// TIA Portal V15.1 export
// export: Created 2026-01-09T13:45:14.0664329Z, ExportSetting WithDefaults, WithReadOnly, DisplayName Totally Integrated Automation Portal, DisplayVersion V15.1 Update 8, DisplayName TIA Portal Openness, DisplayVersion V15.1 Update 8, DisplayName STEP 7 Professional, DisplayVersion V15.1 Update 8, DisplayName WinCC Advanced, DisplayVersion V15.1 Update 8
DATA_BLOCK "C#2_WB"   // DB2
{ S7_Optimized_Access := 'FALSE' }
VERSION : 0.1
// stored: AutoNumber true, CodeModifiedDate 2026-01-04T14:05:19.1281212Z, CompileDate 2026-01-04T14:27:04.768919Z, CreationDate 2024-10-12T12:36:08.0193576Z, DBAccessibleFromOPCUA true, InterfaceModifiedDate 2026-01-04T14:05:19.1281212Z, IsConsistent true, IsKnowHowProtected false, IsOnlyStoredInLoadMemory false, IsPLCDB false, IsWriteProtectedInAS false, ModifiedDate 2026-01-04T14:05:19.1281212Z, ParameterModified 2026-01-04T14:05:19.1281212Z, StructureModified 2026-01-04T14:05:19.1281212Z
   VAR
      F1_NN_RUN : Bool;   // F1 Nút nhấn chạy
      F2_SW_PAU : Bool;   // F2 Công tắc tạm dừng
      F3_NN_STOP : Bool;   // F3 Nút nhấn dừng/hủy mẻ
      F4_SW_SIM : Bool;   // F4 Công tắc chế độ mô phỏng
      "SW_MAN/AUTO" : Bool;   // Công tắc chế độ chạy tay/tự động
      SW_XA_LIEU : Bool;   // Công tắc chế độ xả cân cốt liệu
      SW_NAP_NOI_TRON : Bool;   // Công tắc nạp liệu nồi trộn
      SW_XA_NOI_TRON : Bool;   // Công tắc chế độ xả bê tông
      "NN_NOI TRON" : Bool;   // Nút nhấn Nồi trộn
      NN_BTX : Bool;   // Nút nhấn Băng tải xiên
      NN_BTN : Bool;   // Nút nhấn Băng tải ngang
      "NN_TANG SAY" : Bool;   // Nút nhấn Tang sấy cốt liệu
      "NN_BOM DAU" : Bool;   // Nút nhấn Bơm dầu DO
      "NN_GAU COT LIEU" : Bool;   // Nút nhấn Gàu tải cốt liệu nóng
      "NN_SAN RUNG" : Bool;   // Nút nhấn Sàn rung cốt liệu
      "NN_GAU FD" : Bool;   // Nút nhấn Gàu tải phụ F/D
      "NN_VIT TAI FD" : Bool;   // Nút nhấn Vít tải F/D
      "NN_BOM SBS" : Bool;   // Nút nhấn Bơm nạp hạt nhựa SBS
      "NN_QUAT GIO" : Bool;   // Nút nhấn Quạt gió lọc bụi
      "NN_BOM NUOC" : Bool;   // Nút nhấn Bơm nước lọc bụi
      "NN_MO CUA" : Bool;   // Nút nhấn Van mở cửa nồi trộn
      "NN_DONG CUA" : Bool;   // Nút nhấn Van đóng cửa nồi trộn
      NN_MNK : Bool;   // Nút nhấn Máy nén khí
      "SW_XA CL1" : Bool;   // Công tắc Băng tải xả cốt liệu 1
      "SW_XA CL2" : Bool;   // Công tắc Băng tải xả cốt liệu 2
      "SW_XA CL3" : Bool;   // Công tắc Băng tải xả cốt liệu 3
      "SW_XA CL4" : Bool;   // Công tắc Băng tải xả cốt liệu 4
      "SW_XA CL5" : Bool;   // Công tắc Băng tải xả cốt liệu 5
      "NN_CAN AG1" : Bool;   // Nút nhấn Van cân AG1
      "NN_CAN AG2" : Bool;   // Nút nhấn Van cân AG2
      "NN_CAN AG3" : Bool;   // Nút nhấn Van cân AG3
      "NN_CAN AG4" : Bool;   // Nút nhấn Van cân AG4
      "NN_CAN AG5" : Bool;   // Nút nhấn Van cân AG5
      "NN_CAN FD1" : Bool;   // Nút nhấn Van cân F/D
      "NN_CAN AP1" : Bool;   // Nút nhấn Bơm nhựa
      "NN_CAN SB1" : Bool;   // Nút nhấn Van cân hạt nhựa SBS
      "SW_XA W_AG1" : Bool;   // Công tắc Van xả cân AG1
      "SW_XA W_FD1" : Bool;   // Công tắc Van xả cân FD1
      "SW_XA W_AP1" : Bool;   // Công tắc Van xả cân AP1
      "SW_XA W_SB1" : Bool;   // Công tắc Van xả cân SB1
      "NN_BOM TUOI NHUA" : Bool;   // Nút nhấn Bổ sung 1
      "NN_XA HET AGG" : Bool;   // Nút nhấn Bổ sung 2
      "NN_DAU DOT" : Bool;   // Nút nhấn Bổ sung 3
      NN_VAN_PNSBS : Bool;   // Nút nhấn Bổ sung 4
      "NN_NOTE 5" : Bool;   // Nút nhấn Bổ sung 5
      "NN_NOTE 6" : Bool;   // Nút nhấn Bổ sung 6
      "NN_NOTE 7" : Bool;   // Nút nhấn Bổ sung 7
      NN_FU_AG1 : Bool;   // Nút nhấn Báo đầy silo AG1
      NN_FU_AG2 : Bool;   // Nút nhấn Báo đầy silo AG2
      NN_FU_AG3 : Bool;   // Nút nhấn Báo đầy silo AG3
      NN_FU_AG4 : Bool;   // Nút nhấn Báo đầy silo AG4
      NN_FU_AG5 : Bool;   // Nút nhấn Báo đầy silo AG5
      NN_FU_FD1 : Bool;   // Nút nhấn Báo đầy silo FD1
      NN_FU_AP1 : Bool;   // Nút nhấn Báo đầy silo AP1
      NN_FU_SB1 : Bool;   // Nút nhấn Báo đầy silo SBS1
      SW_PA_AG1 : Bool;   // Công tắc Tạm dừng cân AG1
      SW_PA_AG2 : Bool;   // Công tắc Tạm dừng cân AG2
      SW_PA_AG3 : Bool;   // Công tắc Tạm dừng cân AG3
      SW_PA_AG4 : Bool;   // Công tắc Tạm dừng cân AG4
      SW_PA_AG5 : Bool;   // Công tắc Tạm dừng cân AG5
      SW_PA_FD1 : Bool;   // Công tắc Tạm dừng cân FD1
      SW_PA_AP1 : Bool;   // Công tắc Tạm dừng cân AP1
      SW_PA_SB1 : Bool;   // Công tắc Tạm dừng cân SBS1
      NN_ZERO_AG1 : Bool;   // Nút nhấn chỉnh 0 cân AG1
      NN_SPAN_AG1 : Bool;   // Nút nhấn chỉnh tải cân AG1
      NN_ZERO_FD1 : Bool;   // Nút nhấn chỉnh 0 cân FD1
      NN_SPAN_FD1 : Bool;   // Nút nhấn chỉnh tải cân FD1
      NN_ZERO_AP1 : Bool;   // Nút nhấn chỉnh 0 cân AP1
      NN_SPAN_AP1 : Bool;   // Nút nhấn chỉnh tải cân AP1
      NN_ZERO_SB1 : Bool;   // Nút nhấn chỉnh 0 cân SBS1
      NN_SPAN_SB1 : Bool;   // Nút nhấn chỉnh tải cân SBS1
      "NN_ZERO_TEMP TS" : Bool;   // Nút nhấn chỉnh 0 nhiệt độ 1
      "NN_SPAN_TEMP TS" : Bool;   // Nút nhấn chỉnh tải nhiệt độ 1
      "NN_ZERO_TEMP AG" : Bool;   // Nút nhấn chỉnh 0 nhiệt độ 2
      "NN_SPAN_TEMP AG" : Bool;   // Nút nhấn chỉnh tải nhiệt độ 2
      "NN_ZERO_TEMP AP" : Bool;   // Nút nhấn chỉnh 0 nhiệt độ 3
      "NN_SPAN_TEMP AP" : Bool;   // Nút nhấn chỉnh tải nhiệt độ 3
      "NN_ZERO_TEMP TL" : Bool;   // Nút nhấn chỉnh 0 nhiệt độ 4
      "NN_SPAN_TEMP TL" : Bool;   // Nút nhấn chỉnh tải nhiệt độ 4
      "NN_RUNG AG1" : Bool;   // Nút nhấn rung phễu cân AG1
      "NN_RUNG FD1" : Bool;   // Nút nhấn rung phễu cân FD1
      "NN_RUNG SB1" : Bool;   // Nút nhấn rung phễu cân SBS1
      "XAC NHAN CAN DU" : Bool;   // Nút nhấn xác nhận cân dư
      XNC_AUT_AG1 : Bool;   // Tự dộng xác nhận cân dư Agg1
      XNC_AUT_AG2 : Bool;   // Tự dộng xác nhận cân dư Agg2
      XNC_AUT_AG3 : Bool;   // Tự dộng xác nhận cân dư Agg3
      XNC_AUT_AG4 : Bool;   // Tự dộng xác nhận cân dư Agg4
      XNC_AUT_AG5 : Bool;   // Tự dộng xác nhận cân dư Agg5
      XNC_AUT_FD1 : Bool;   // Tự dộng xác nhận cân dư FD1
      XNC_AUT_AP1 : Bool;   // Tự dộng xác nhận cân dư AP1
      XNC_AUT_SB1 : Bool;   // Tự dộng xác nhận cân dư SBS1
      BUTRU_AGG1 : Bool;   // Bù trừ khối lượng Agg1
      BUTRU_AGG2 : Bool;   // Bù trừ khối lượng Agg2
      BUTRU_AGG3 : Bool;   // Bù trừ khối lượng Agg3
      BUTRU_AGG4 : Bool;   // Bù trừ khối lượng Agg4
      BUTRU_AGG5 : Bool;   // Bù trừ khối lượng Agg5
      BUTRU_FD1 : Bool;   // Bù trừ khối lượng FD1
      BUTRU_AP1 : Bool;   // Bù trừ khối lượng AP1
      BUTRU_SB1 : Bool;   // Bù trừ khối lượng SBS1
      "NN_RUNG CL1" : Bool;
      "NN_RUNG CL2" : Bool;
      "NN_RUNG CL3" : Bool;
      SETUP_MODE_DOC_LAP : Bool;   // OFF=cộng dồn, ON=độc lập
      NN_ZERO_IND_AG1 : Bool;
      NN_SPAN_IND_AG1 : Bool;
      NN_ZERO_IND_AG2 : Bool;
      NN_SPAN_IND_AG2 : Bool;
      NN_ZERO_IND_AG3 : Bool;
      NN_SPAN_IND_AG3 : Bool;
      NN_ZERO_IND_AG4 : Bool;
      NN_SPAN_IND_AG4 : Bool;
      NN_ZERO_IND_AG5 : Bool;
      NN_SPAN_IND_AG5 : Bool;
   END_VAR
BEGIN
END_DATA_BLOCK
